Staubli VAL3: countBits.pgx

program countBits(lists& x_lInput[], num& x_nResult[])
  local num l_nElement
  local num l_nBits
begin

  resize(x_nResult,1,1)
  x_nResult[0] = 0
  resize(x_nResult,1,12)

  for l_nBits = 0 to 11
    for l_nElement = 0 to size(x_lInput)-1
      call util:vec2num(x_lInput[l_nElement].sString[l_nBits], nNum)
      x_nResult[l_nBits] = x_nResult[l_nBits] + nNum
    endFor
  endFor


end
